FUNCTION_BLOCK ILOCK_CONFLICT_TRIP_A2X (* Prioritizes the first active input and trips on conflict. Requires RESET (Adapter Version, UP/DOWN fed from a single A2X input/output). *)
  (* Standard: 61499-2; Description: Copyright (c) 2026 HR Agrartechnik GmbH This program and the accompanying materials are made available under the terms of the Eclipse Public License 2.0 which is available at https://www.eclipse.org/legal/epl-2.0/ SPDX-License-Identifier: EPL-2.0 *)
  (* Version 1.0, 2026-09-05, Franz Höpfinger, HR Agrartechnik GmbH, initial API and implementation and/or initial documentation *)
  PACKAGE logiBUS::signalprocessing::interlock;
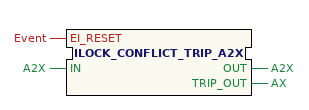
  EVENT_INPUT
    EI_RESET;
  END_EVENT
  SOCKETS
    IN : adapter::types::unidirectional::A2X; (* Input for forward/up and backward/down direction *)
  END_SOCKETS
  PLUGS
    OUT : adapter::types::unidirectional::A2X; (* Output for forward/up and backward/down direction *)
    TRIP_OUT : adapter::types::unidirectional::AX; (* Trip State Output *)
  END_PLUGS
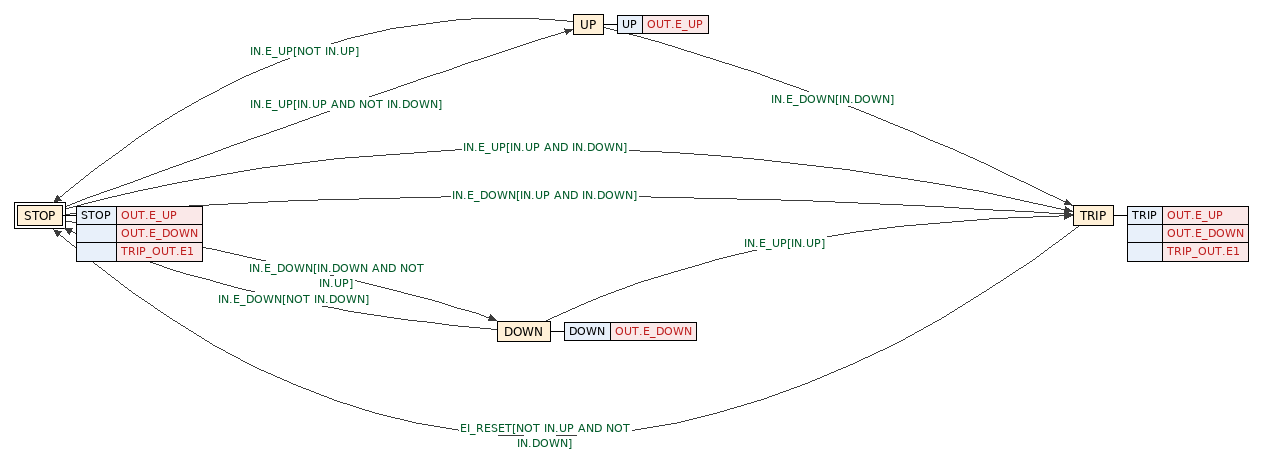
  EC_STATES
    STOP : STOP -> OUT.E_UP, -> OUT.E_DOWN, -> TRIP_OUT.E1;
    UP : UP -> OUT.E_UP;
    DOWN : DOWN -> OUT.E_DOWN;
    TRIP : TRIP -> OUT.E_UP, -> OUT.E_DOWN, -> TRIP_OUT.E1;
  END_STATES
  EC_TRANSITIONS
    STOP TO UP := IN.E_UP[IN.UP AND NOT IN.DOWN];
    STOP TO DOWN := IN.E_DOWN[IN.DOWN AND NOT IN.UP];
    STOP TO TRIP := IN.E_UP[IN.UP AND IN.DOWN];
    STOP TO TRIP := IN.E_DOWN[IN.UP AND IN.DOWN];
    UP TO STOP := IN.E_UP[NOT IN.UP];
    UP TO TRIP := IN.E_DOWN[IN.DOWN];
    DOWN TO STOP := IN.E_DOWN[NOT IN.DOWN];
    DOWN TO TRIP := IN.E_UP[IN.UP];
    TRIP TO STOP := EI_RESET[NOT IN.UP AND NOT IN.DOWN];
  END_TRANSITIONS
  ALGORITHM UP IN ST:
OUT.UP := BOOL#TRUE;
OUT.DOWN := BOOL#FALSE;
TRIP_OUT.D1 := BOOL#FALSE;
  END_ALGORITHM
  ALGORITHM DOWN IN ST:
OUT.UP := BOOL#FALSE;
OUT.DOWN := BOOL#TRUE;
TRIP_OUT.D1 := BOOL#FALSE;
  END_ALGORITHM
  ALGORITHM STOP IN ST:
OUT.UP := BOOL#FALSE;
OUT.DOWN := BOOL#FALSE;
TRIP_OUT.D1 := BOOL#FALSE;
  END_ALGORITHM
  ALGORITHM TRIP IN ST:
OUT.UP := BOOL#FALSE;
OUT.DOWN := BOOL#FALSE;
TRIP_OUT.D1 := BOOL#TRUE;
  END_ALGORITHM
END_FUNCTION_BLOCK
